TYPE INTERNAL ST_CylinderConfig :
STRUCT
	delayTimeAfterReachedHP		: TIME;
	delayTimeAfterReachedWP		: TIME;
	movementTimeout				: TIME:= T#5S;
	monitorSensorsOverlap		: BOOL:= TRUE;
	sensorsOverlapTimeout		: TIME:= T#100MS;
END_STRUCT
END_TYPE

(* stored: Version 1.1.0.1, ProductVersion 3.1.4026.17
   DUT ST_CylinderConfig: Id {51cf3f94-4ba8-0b5b-3c59-374576c52871} *)
